TYPE STATE:
    STRUCT
        curTime: REAL;
        dvar_M_p_v0: REAL;
        dvar_M_p_v1: DINT;
        dvar_M_p_v2: DINT;
        dvar_M_p_v3: DINT;
        dvar_M_p_v99: REAL;
        dvar_M_p_vx: REAL;
        dvar_M_p_vr: TupleStruct_1;
        dvar_M_p: DINT;
    END_STRUCT;
END_TYPE
